// TIA Portal V18 export
VAR_GLOBAL   // PLC tag table "tag"
   input AT %I0.0 : Bool;
   output AT %Q0.0 : Bool;
   memory AT %M0.0 : Bool;
   salida AT %Q0.1 : Bool;
   entrada AT %I0.2 : Bool;
   ent AT %I0.3 : Bool;
END_VAR
